{attribute 'GeneratedUsingTerminal: EK1100-0000-0018'}
{attribute addProperty BoxType "EK1100-0000-0018"}
{attribute addProperty Id "Beckhoff_ER4xxxEK1122Beckhoff_ER4xxxEK1122_B7F32B36112"}
{attribute addProperty CRC "3090179415"}
{attribute addProperty Size "112"}
TYPE Beckhoff_ER4xxx_B8306557 EXTENDS EK1100_1FC0878B :
STRUCT
	{attribute addProperty Name "Beckhoff_ER4xxxEK1122"}
	{attribute addProperty PreviousPort "Beckhoff ER4xxx : B"}
	Beckhoff_ER4xxxEK1122 : Beckhoff_ER4xxxEK1122_B7F32B36;
END_STRUCT
END_TYPE

(* stored: Version 1.2.0.0, ProductVersion 3.1.4024.9
   DUT Beckhoff_ER4xxx_B8306557: Id {c62ce99a-fb1d-4dc0-b815-96cfd55bac89} *)
